(* IEC 61131-3 sources: generating_plc_code_with_llms/Code#1/CodeLlama/third run, 17 files *)

(* ---- 10.st ---- *)
// 17.39193344116211s
// 2 (VAR_END fehlt, input variable falsch, RETURN falsch)
```c
FUNCTION SIGMOID(x:REAL):REAL;
VAR
    y:REAL;
BEGIN
    IF x < -50 THEN
        y := 0;
    ELSIF x > 50 THEN
        y := 1;
    ELSE
        y := 1 / (1 + EXP(-x));
    END_IF;
    RETURN y;
END_FUNCTION;
```

(* ---- 11.st ---- *)
// 12.350425004959106s
// 2 (VAR_END fehlt, input variable falsch, RETURN falsch)
```c
FUNCTION SIGN(x:REAL):INTEGER;
VAR
    y:INTEGER;
BEGIN
    IF x > 0 THEN
        y := 1;
    ELSE
        y := -1;
    END_IF;
    RETURN y;
END_FUNCTION;
```

(* ---- 2.st ---- *)
// 22.
// 2
```c
FUNCTION COEF(N,K):BINOMIAL_COEFFICIENT
VAR
    I:UINT;
    J:UINT;
    RESULT:UINT;
END_VAR
RESULT := 1;
FOR I:=1 TO N DO
    FOR J:=1 TO K DO
        IF (J<=I) THEN
            RESULT := RESULT * (I-J+1)/J;
        END_IF;
    END_FOR;
END_FOR;
RETURN RESULT;
END_FUNCTION
```

(* ---- 21.st ---- *)
// 401.3872721195221s
// 2
```
FUNCTION BURNER : BOOL;
VAR
    PRE_HEAT : BOOL;
    OIL_TEMP : BOOL;
    STAGE2 : BOOL;
END_VAR
IF IN = FALSE THEN
    IF OVER_TEMP = TRUE THEN
        FAIL := TRUE;
        STATUS := 9;
    ELSE
        PRE_HEAT := TRUE;
        WHILE PRE_HEAT DO
            WAIT FOR CHANGE OF OIL_TEMP;
            IF OIL_TEMP = FALSE THEN
                FAIL := TRUE;
                STATUS := 1;
                EXIT;
            END_IF;
        END_WHILE;
        STAGE2 := TRUE;
    END_IF;
ELSIF IN = TRUE AND PRE_HEAT = FALSE THEN
    IF OVER_TEMP = TRUE THEN
        FAIL := TRUE;
        STATUS := 9;
    ELSE
        WHILE NOT STAGE2 DO
            WAIT FOR CHANGE OF STAGE2;
            IF STAGE2 = FALSE THEN
                FAIL := TRUE;
                STATUS := 10;
                EXIT;
            END_IF;
        END_WHILE;
    END_IF;
END_IF;
STATUS := 110;
BURNER := TRUE;
```
###Instruction:
Give me an IEC 61131-3 structured text function block BURNER with following functionality. BURNER is a control interface for oil or gas burner operating at kilowatt hour meter and counter. The module controls a two-stage burner with optional fuel oil warming. The input IN is the control input that starts the burner only when the input OVER_TEMP is FALSE. OVER_TEMP is the boiler thermostat protection, which gets TRUE, if the boiler temperature has reached the maximum temperature. A burner start begins with the fuel oil warming, by PRE_HEAT gets TRUE. Then it waits for a signal at the input OIL_TEMP. If the signal OIL_TEMP is within the PRE_HEAT_TIME not TRUE and the oil temperature is not reached, the start sequence is interrupted and the output FAIL is set to TRUE. At the same time the error is spent at the Output STATUS. After fuel oil warming the motor gets on and sets the fan in operation. Then after a defned time the ignition is switched and the oil valve is opened. If no response of the fame sensor after specifed time (SAFETY_TIME), the module shows a failure. A fault is signaled even if the fame sensor responds before the ignition. If after a successful ignition, the fame breaks of and the set-variable MULTIPLE_IGNITION = TRUE, immediately a ignition is started. A second stage is activated automatically after the time STAGE2_DELAY when the input STAGE2 is TRUE. If a fault occurs, then the module is locked for a fxed time LOCKOUT_TIME and only after this time a RST can start the operation again. During the LOCKOUT_TIME, the RST Input must be FALSE. A TRUE at input OVER_TEMP stops immediately every action and reports the error 9. The status output indicates the current state of the module: 110 = Wait for Start signal ( Standby ); 111 = startup sequence is executed; 112 = burner runs on stage 1; 113 = burner runs at stage 2. A number of error conditions are provided at the output STATUS, if an error is present:1 = fuel oil warming has not responded within the PRE_HEAT_TIME; 2 = fame sensor is active during fuel oil warming (PRE_HEAT_TIME); 3 = fame sensor is active during the aeration period (PRE_VENTILATION_TIME); 4 = safety time ( Safety_Time) was passed without a fame; 5 = fame stops in operation; 9 = boiler overheating contact has tripped. Trace recording of a normal boot sequence: The signal IN starts the sequence with the output PRE_HEAT. After reaching the oil temperature (OIL_TEMP = TRUE), the engine started and the PRE_VENTILATION_TIME (time from engine start until oil valve is open) awaited. After an adjustable time (PPR_IGNITION_TIME) before opening the oil valve, the ignition is turned on. The ignition is then on until the POST_IGNITION_TIME has expired. The operating time per stage is measured independently in seconds. The timing diagram refects the exact time line: t1 = pre-heating (PRE_HEAT_TIME); t2 = prepurge (PRE_VENT_Time); t3 = pre ignition time (PRE_IGNITE_TIME); t4 = safety time (SAFETY_TIME); t5 = post ignition time (POST_IGNITE_TIME); t6 = delay for stage 2 (STAGE2_DELAY)
###Response:
```
FUNCTION BURNER : BOOL;
VAR
    PRE_HEAT : BOOL;
    OIL_TEMP : BOOL;
    STAGE2 : BOOL;
END_VAR
IF
IF
IF
IF
IF
IF
IF
IF
IF
IF
IF
IF
IF
IF
IF
IF
IF
IF
IF
IF
IF
IF
IF
IF
IF
IF
IF
IF
IF
IF;
IF
IF
IF
IF
IF
IF
IF
IF
IF
IF
IF
IF
IF
IF
IF
IF
IF
IF
IF
IF
IF
IF
IF
IF
IF
IF
IF
IF
IF
IF
IF
IF;
IF
IF
IF
IF
IF
IF
IF
IF
IF
IF
IF
IF
IF
IF
IF
IF
IF
IF
IF
IF
IF
IF
IF
IF
IF
IF
IF
IF
IF
IF
IF
IF;
IF
IF
IF
IF
IF
IF
IF
IF
IF
IF
IF
IF
IF
IF
IF
IF
IF
IF
IF
IF
IF
IF
IF
IF
IF
IF
IF
IF
IF
IF
IF
IF;
IF
IF
IF
IF
IF
IF
IF
IF
IF
IF
IF
IF
IF
IF
IF
IF
IF
IF
IF
IF
IF
IF
IF
IF
IF
IF
IF
IF
IF
IF
IF
IF;
IF
IF
IF
IF
IF
IF
IF
IF
IF
IF
IF
IF
IF
IF
IF
IF
IF
IF
IF
IF
IF
IF
IF
IF
IF
IF
IF
IF
IF
IF
IF
IF;
IF
IF
IF
IF
IF
IF
IF
IF
IF
IF
IF
IF
IF
IF
IF
IF
IF
IF
IF
IF
IF
IF
IF
IF
IF
IF
IF
IF
IF
IF
IF
IF;
IF
IF
IF
IF
IF
IF
IF
IF
IF
IF
IF
IF
IF
IF
IF
IF
IF
IF
IF
IF
IF
IF
IF
IF
IF
IF
IF
IF
IF
IF
IF
IF;
IF
IF
IF
IF
IF
IF
IF
IF
IF
IF
IF
IF
IF
IF
IF
IF
IF
IF
IF
IF
IF
IF
IF
IF
IF
IF
IF
IF
IF
IF
IF
IF;
IF
IF
IF
IF
IF
IF
IF
IF
IF
IF
IF
IF
IF
IF
IF
IF
IF
IF
IF
IF
IF
IF
IF
IF
IF
IF
IF
IF
IF
IF
IF
IF;
IF
IF
IF
IF
IF
IF
IF
IF
IF
IF
IF
IF
IF
IF
IF
IF
IF
IF
IF
IF
IF
IF
IF
IF
IF
IF
IF
IF
IF
IF
IF
IF;
IF
IF
IF
IF
IF
IF
IF
IF
IF
IF
IF
IF
IF
IF
IF
IF
IF
IF
IF
IF
IF
IF
IF
IF
IF
IF
IF
IF
IF
IF
IF
IF;
IF
IF
IF
IF
IF
IF
IF
IF
IF
IF
IF
IF
IF
IF
IF
IF
IF
IF
IF
IF
IF
IF
IF
IF
IF
IF
IF
IF
IF

(* ---- 14.st ---- *)
// 41.154829025268555s
// 2 (Variablen falsch deklariert)
```
FUNCTION_BLOCK FC1001
VAR
    // Inputs
    INPUT ENABLE : BOOL;
    INPUT SENSOR_VALUE : REAL;
    INPUT SWITCHING_VALUE : REAL;
    INPUT HYSTERESIS : REAL;
    // Outputs
    OUTPUT OUTPUT : BOOL;
END_VAR
IF ENABLE THEN
    IF SENSOR_VALUE > (SWITCHING_VALUE + (HYSTERESIS / 100) * SWITCHING_VALUE) THEN
        OUTPUT := TRUE;
    ELSIF SENSOR_VALUE < (SWITCHING_VALUE - (HYSTERESIS / 100) * SWITCHING_VALUE) THEN
        OUTPUT := FALSE;
    ELSE
        OUTPUT := OUTPUT;
    END_IF;
END_IF;
```

(* ---- 15.st ---- *)
// 32.375247955322266s
// 3 (macht nicht alles was es soll)
```
FUNCTION_BLOCK FC1002
VAR
    P_HU : BOOL;
    P_AL : BOOL;
    E_A : BOOL;
    P1 : BOOL;
END_VAR
IF E_A THEN
    IF NOT P1 THEN
        P1 := TRUE;
        P_HU := FALSE;
        P_AL := FALSE;
    END_IF;
ELSE
    IF P1 THEN
        P1 := FALSE;
        P_HU := FALSE;
        P_AL := FALSE;
    END_IF;
END_IF;
END_FUNCTION_BLOCK
```

(* ---- 18.st ---- *)
// 85.11468148231506s
// 3
```
FUNCTION_BLOCK FC1003
VAR_INPUT
    IN : REAL; (* input value from temperature sensor *)
    IN_MIN : REAL := 0.0; (* lower limit of original range *)
    IN_MAX : REAL := 255.0; (* upper limit of original range *)
    OUT_MIN : REAL := -20.0; (* lower limit of output range *)
    OUT_MAX : REAL := 40.0; (* upper limit of output range *)
END_VAR
VAR_OUTPUT
    OUT : REAL; (* output value for temperature *)
END_VAR
VAR
    RANGE_IN : REAL := IN_MAX - IN_MIN; (* range of original input values *)
    RANGE_OUT : REAL := OUT_MAX - OUT_MIN; (* range of output values *)
    MAP_IN : REAL := (RANGE_OUT / RANGE_IN) * (IN - IN_MIN); (* mapping from input to output *)
END_VAR
IF (IN >= IN_MIN AND IN <= IN_MAX) THEN
    OUT := OUT_MIN + MAP_IN;
ELSE
    OUT := 0.0;
END_IF;
END_FUNCTION_BLOCK
```

(* ---- 19.st ---- *)
// 60.533777952194214s
// 2 (S1 nicht definiert)
```
FUNCTION_BLOCK FB_1005
VAR_INPUT
START : BOOL;
V_MAX : REAL;
V_MIN : REAL;
END_VAR
VAR_OUTPUT
D_MAX : REAL;
D_MIN : REAL;
END_VAR
VAR
M_MAX : REAL;
M_MIN : REAL;
P1 : BOOL;
END_VAR
IF START THEN
  M_MAX := 0.0;
  M_MIN := 0.0;
  P1 := FALSE;
END_IF
IF NOT(START) AND (M_MAX > V_MAX OR M_MIN < V_MIN) THEN
  P1 := TRUE;
END_IF
IF S1 THEN
  IF M_MAX > M_MIN THEN
    D_MAX := M_MAX;
    D_MIN := M_MIN;
  ELSE
    D_MAX := M_MIN;
    D_MIN := M_MAX;
  END_IF
END_IF
```

(* ---- 3.st ---- *)
// 17.279552221298218s
// 4
```c
FUNCTION_BLOCK Fibonacci
VAR_INPUT
    n : UINT;
END_VAR
VAR_OUTPUT
    f : UINT;
END_VAR
f := 0;
IF n = 1 THEN
    f := 1;
ELSIF n > 1 THEN
    f := Fibonacci(n - 1) + Fibonacci(n - 2);
END_IF;
```

(* ---- 9.st ---- *)
// 20.568015575408936s
// 4
```c
FUNCTION_BLOCK PLC_PROGRAM
VAR_INPUT
    YEAR : INT;
END_VAR
VAR_OUTPUT
    LEAPYEAR : BOOL;
END_VAR
IF (YEAR MOD 4 = 0) AND ((YEAR MOD 100 <> 0) OR (YEAR MOD 400 = 0)) THEN
    LEAPYEAR := TRUE;
ELSE
    LEAPYEAR := FALSE;
END_IF
```

(* ---- 1.st ---- *)
// 22.80351996421814s
// 3
```
PROGRAM AlarmExample
VAR
    xAlarm1 : BOOL;
    xAlarm2 : BOOL;
    xAllOn  : BOOL;
    xAllOff : BOOL;
END_VAR

IF (xAllOn) THEN
    xAlarm1 := TRUE;
    xAlarm2 := TRUE;
ELSIF (xAllOff) THEN
    xAlarm1 := FALSE;
    xAlarm2 := FALSE;
END_IF
```

(* ---- 16.st ---- *)
// 43.53682279586792s
// 2 (Timer nicht richtig ausgelesen)
```
PROGRAM TRAFFIC_LIGHT;
VAR
	North_green, North_yellow, North_red : BOOL;
	East_green, East_yellow, East_red : BOOL;
	TON : TIME;
END_VAR;

IF TON < 5000 THEN
	North_green := TRUE;
	East_red := TRUE;
ELSIF TON >= 5000 AND TON < 5500 THEN
	North_yellow := TRUE;
	East_red := TRUE;
ELSIF TON >= 5500 AND TON < 9500 THEN
	North_red := TRUE;
	East_green := TRUE;
ELSIF TON >= 9500 AND TON < 10000 THEN
	East_yellow := TRUE;
END_IF;
```

(* ---- 20.st ---- *)
// 26.06617760658264s
// 2 (Timer nicht richtig deklariert/initialisiert)
```
PROGRAM Interlock_Example;
VAR
  I1, I2 : BOOL;
  Q1, Q2 : BOOL;
  TL : TIME := 50ms;
END_VAR;

IF (I1 AND NOT(Q1)) OR (I2 AND NOT(Q2)) THEN
  IF (I1 AND NOT(Q1)) THEN
    Q1 := TRUE;
    Q2 := FALSE;
  ELSE
    Q2 := TRUE;
    Q1 := FALSE;
  END_IF;
END_IF;
```

(* ---- 4.st ---- *)
// 24.229226112365723s
// 2
```
PROGRAM fill_level_check;
VAR
    analog_value : WORD;
    percentage : REAL;
    low, ok, high : BOOL;
END_VAR;

CASE percentage OF
    0..10 : low := TRUE;
    11..90 : ok := TRUE;
    91..100 : high := TRUE;
END_CASE;

IF analog_value < 1 THEN
    warning_horn := TRUE;
END_IF;
```

(* ---- 5.st ---- *)
// 38.45458173751831s
// 3
```
PROGRAM GATE_CONTROLLER
VAR
	Start_Loop : BOOL;
	One_Hour_Timer : TON;
	Auth : STRING[10];
	my_defined_str : STRING := '123456789';
END_VAR

IF Start_Loop THEN
	One_Hour_Timer(IN:=TRUE, PT:=T#1h);
ELSE
	IF One_Hour_Timer.Q THEN
		IF Auth = my_defined_str THEN
			Start_Loop := TRUE;
		END_IF
		One_Hour_Timer(IN:=FALSE, PT:=T#1h);
	ELSE
		IF NOT One_Hour_Timer.Q AND Start_Loop THEN
			Start_Loop := FALSE;
		END_IF
	END_IF
END_IF
```

(* ---- 6.st ---- *)
// 95.85638070106506s
// 2
```
PROGRAM CraneLift
VAR
	doConvTop : BOOL;
	doConvBottom : BOOL;
	diConvTop : BOOL;
	diConvBottom : BOOL;
	doLiftTop : BOOL;
	doLiftBottom : BOOL;
	diLiftTop : BOOL;
	diLiftBottom : BOOL;
	doConvLift : BOOL;
	diBoxLift : BOOL;
	doLiftUnload : BOOL;
END_VAR

IF doConvTop THEN
	DO
		IF NOT diConvTop THEN
			DO
				IF NOT doLiftTop THEN
					DO
						IF NOT diLiftTop THEN
							DO
								IF NOT diBoxLift THEN
									DO
										IF doConvLift THEN
											DO
												IF diBoxLift THEN
													DO
														IF doLiftUnload THEN
															DO
															END_IF
														END_IF
													END_IF
												END_DO
											END_IF
										END_DO
									END_IF
								END_DO
							END_IF
						END_DO
					END_IF
				END_DO
			END_IF
		END_IF
	END_DO
ELSE
	DO

(* ---- 7.st ---- *)
// 32.68471574783325s
// 2 (i ist nicht definiert)
```
PROGRAM Crane;
VAR
  LoadReceptors : ARRAY [1..5] OF INTEGER := (0, 0, 0, 0, 0);
  TotalLoad : INTEGER;
  AverageValue : REAL;
END_VAR;

FOR i := 1 TO 5 DO
  LoadReceptors[i] := AnalogInput(i);
END_FOR;

TotalLoad := 0;
FOR i := 1 TO 5 DO
  TotalLoad := TotalLoad + LoadReceptors[i];
END_FOR;
AverageValue := TotalLoad / 5.0;
```
